// Mitsubishi GX Works2 project: LuuVT   PLC: FX3U/FX3UC

PROGRAM MAIN
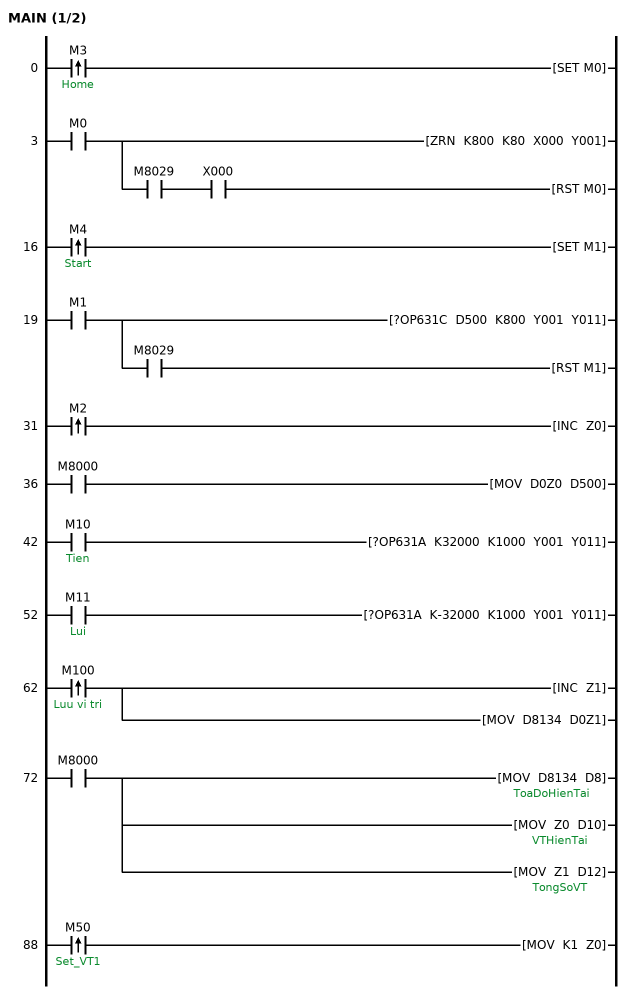
0     LDP     M3  ; Home
      SET     M0
3     LD      M0
      ZRN     K800 K80 X000 Y001
      AND     M8029
      AND     X000
      RST     M0
16    LDP     M4  ; Start
      SET     M1
19    LD      M1
      ?OP631C D500 K800 Y001 Y011
      AND     M8029
      RST     M1
31    LDP     M2
      INC     Z0
36    LD      M8000
      MOV     D0Z0 D500
42    LD      M10  ; Tien
      ?OP631A K32000 K1000 Y001 Y011
52    LD      M11  ; Lui
      ?OP631A K-32000 K1000 Y001 Y011
62    LDP     M100  ; Luu vi tri
      INC     Z1
      MOV     D8134 D0Z1
72    LD      M8000
      MOV     D8134 D8  ; ToaDoHienTai
      MOV     Z0 D10  ; VTHienTai
      MOV     Z1 D12  ; TongSoVT
88    LDP     M50  ; Set_VT1
      MOV     K1 Z0
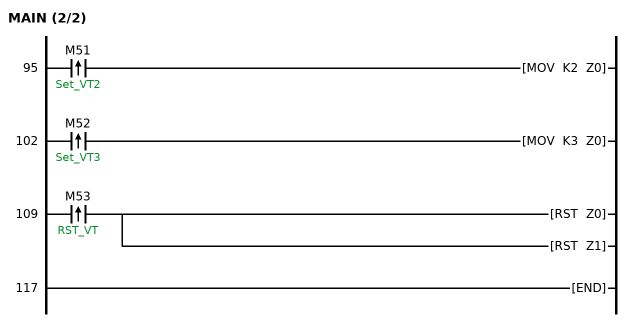
95    LDP     M51  ; Set_VT2
      MOV     K2 Z0
102   LDP     M52  ; Set_VT3
      MOV     K3 Z0
109   LDP     M53  ; RST_VT
      RST     Z0
      RST     Z1
117   END
END_PROGRAM

// device comments not shown above
D1  ; ViTri1
D2  ; ViTri2
D3  ; ViTri3
